
// ===== library: MasterCopy "enkoder_okuma" =====

FUNCTION_BLOCK "enkoder_okuma"   // FB1, LAD
{ S7_Optimized_Access := 'TRUE' }
VERSION : 0.1
   VAR_INPUT
      ENKODER_GELEN_PULSE : UInt;
      ENKODER_PULSE_COZUNURLUGU : LInt;
   END_VAR
   VAR_OUTPUT
      DERECE_FARKI : DInt;
   END_VAR
   VAR RETAIN
      mevcut_pulse : UDInt;
      sonraki_pulse : Real;
   END_VAR
   VAR
      pulse_farki : Real;
   END_VAR
   VAR RETAIN
      onceki_pulse : Real;
      NORM_XX : Real;
      NORM_4 : Real;
      mevcut_derece : DInt;
      sonraki_derece : UDInt;
      onceki_derece : UDInt;
   END_VAR
BEGIN

REGION Network 1 (SCL)

   #mevcut_pulse :=#ENKODER_GELEN_PULSE;

   #sonraki_derece := #mevcut_derece;

   #DERECE_FARKI := #sonraki_derece - #onceki_derece;

   IF #DERECE_FARKI < -1000 THEN

       #DERECE_FARKI:= #sonraki_derece + 6975 - #onceki_derece;

   END_IF;

   #sonraki_pulse := #mevcut_pulse;

   #pulse_farki := #sonraki_pulse -#onceki_pulse;

   IF #pulse_farki > 32000 THEN

       #pulse_farki := #onceki_pulse + 65536 - #sonraki_pulse;

   END_IF;

   IF #pulse_farki < -32000 THEN

       #pulse_farki := #sonraki_pulse + 65536 - #onceki_pulse;

   END_IF;

   #NORM_XX += #pulse_farki;

   IF #NORM_XX >= 122880 THEN

       #NORM_XX := 0;

   END_IF;


   #NORM_4 := NORM_X(MIN := 0, VALUE := #NORM_XX, MAX := #ENKODER_PULSE_COZUNURLUGU);

   #mevcut_derece := SCALE_X(MIN := 0, VALUE := #NORM_4, MAX := 360);

   //
   // Enkoder mili ile sistem arasında redüktör var ise ->
   //#mevcut_derece *= 31;
   //#mevcut_derece /= 24;
   //

   #onceki_derece := #sonraki_derece;

   #onceki_pulse := #sonraki_pulse;
END_REGION
END_FUNCTION_BLOCK